LIN {X 0,Y 105.246,Z 1223.954,A -85,B 0,C 180,E1 5404.905,E2 5404.905} C_VEL
LIN {X 0,Y 105.222,Z 1230.827,A -85,B 0,C 180,E1 5396.186,E2 5396.186} C_VEL
LIN {X 0,Y 106.17,Z 1236.984,A -85,B 0,C 180,E1 5386.937,E2 5386.937} C_VEL
LIN {X 0,Y 110.756,Z 1244.43,A -85,B 0,C 180,E1 5373.745,E2 5373.745} C_VEL
LIN {X 0,Y 122.979,Z 1251.855,A -85,B 0,C 180,E1 5359.424,E2 5359.424} C_VEL
LIN {X 0,Y 127.608,Z 1253.595,A -85,B 0,C 180,E1 5355.812,E2 5355.812} C_VEL
LIN {X 0,Y 113.507,Z 1251.143,A -85,B 0,C 180,E1 5342.256,E2 5342.256} C_VEL
LIN {X 0,Y 107.747,Z 1247.277,A -85,B 0,C 180,E1 5327.84,E2 5327.84} C_VEL
LIN {X 0,Y 107.702,Z 1242.807,A -85,B 0,C 180,E1 5316.404,E2 5316.404} C_VEL
LIN {X 0,Y 108.21,Z 1239.966,A -85,B 0,C 180,E1 5311.066,E2 5311.066} C_VEL
LIN {X 0,Y 107.704,Z 1235.764,A -85,B 0,C 180,E1 5305.214,E2 5305.214} C_VEL
LIN {X 0,Y 106.691,Z 1233.424,A -85,B 0,C 180,E1 5296.458,E2 5296.458} C_VEL
LIN {X 0,Y 107.812,Z 1229.194,A -85,B 0,C 180,E1 5287.083,E2 5287.083} C_VEL
LIN {X 0,Y 111.454,Z 1223,A -85,B 0,C 180,E1 5278.05,E2 5278.05} C_VEL
LIN {X 0,Y 117.077,Z 1215.245,A -85,B 0,C 180,E1 5270.178,E2 5270.178} C_VEL
LIN {X 0,Y 124.096,Z 1206.072,A -85,B 0,C 180,E1 5263.528,E2 5263.528} C_VEL
LIN {X 0,Y 128.676,Z 1200.056,A -85,B 0,C 180,E1 5260.161,E2 5260.161} C_VEL
LIN {X 0,Y 131.324,Z 1195.46,A -85,B 0,C 180,E1 5257.692,E2 5257.692} C_VEL
LIN {X 0,Y 135.926,Z 1183.249,A -85,B 0,C 180,E1 5251.112,E2 5251.112} C_VEL
LIN {X 0,Y 138.939,Z 1177.877,A -85,B 0,C 180,E1 5249.119,E2 5249.119} C_VEL
LIN {X 0,Y 147.608,Z 1163.811,A -85,B 0,C 180,E1 5245.692,E2 5245.692} C_VEL
LIN {X 0,Y 155.785,Z 1148.222,A -85,B 0,C 180,E1 5242.936,E2 5242.936} C_VEL
LIN {X 0,Y 162.689,Z 1132.349,A -85,B 0,C 180,E1 5240.917,E2 5240.917} C_VEL
LIN {X 0,Y 168.161,Z 1116.222,A -85,B 0,C 180,E1 5239.397,E2 5239.397} C_VEL
LIN {X 0,Y 172.478,Z 1099.347,A -85,B 0,C 180,E1 5238.341,E2 5238.341} C_VEL
LIN {X 0,Y 175.176,Z 1083.244,A -85,B 0,C 180,E1 5237.612,E2 5237.612} C_VEL
LIN {X 0,Y 175.933,Z 1079.237,A -85,B 0,C 180,E1 5237.531,E2 5237.531} C_VEL
LIN {X 0,Y 193.961,Z 1045.169,A -85,B 0,C 180,E1 5234.022,E2 5234.022} C_VEL
LIN {X 0,Y 205.367,Z 1022.293,A -85,B 0,C 180,E1 5232.228,E2 5232.228} C_VEL
LIN {X 0,Y 209.325,Z 993.562,A -85,B 0,C 180,E1 5227.548,E2 5227.548} C_VEL
LIN {X 0,Y 214.843,Z 962.441,A -85,B 0,C 180,E1 5223.335,E2 5223.335} C_VEL
LIN {X 0,Y 220.959,Z 932.764,A -85,B 0,C 180,E1 5220.051,E2 5220.051} C_VEL
LIN {X 0,Y 225.837,Z 909.225,A -85,B 0,C 180,E1 5217.843,E2 5217.843} C_VEL
LIN {X 0,Y 221.843,Z 897.978,A -85,B 0,C 180,E1 5214.05,E2 5214.05} C_VEL
LIN {X 0,Y 217.917,Z 887.098,A -85,B 0,C 180,E1 5209.959,E2 5209.959} C_VEL
LIN {X 0,Y 214.165,Z 877.016,A -85,B 0,C 180,E1 5205.674,E2 5205.674} C_VEL
LIN {X 0,Y 210.547,Z 867.306,A -85,B 0,C 180,E1 5200.905,E2 5200.905} C_VEL
LIN {X 0,Y 208.954,Z 871.161,A -85,B 0,C 180,E1 5200.494,E2 5200.494} C_VEL
LIN {X 0,Y 201.666,Z 897.41,A -85,B 0,C 180,E1 5198.009,E2 5198.009} C_VEL
LIN {X 0,Y 201.281,Z 903.477,A -85,B 0,C 180,E1 5197.701,E2 5197.701} C_VEL
LIN {X 0,Y 187.356,Z 1041.59,A -85,B 0,C 180,E1 5194.545,E2 5194.545} C_VEL
LIN {X 0,Y 184.433,Z 1072.002,A -85,B 0,C 180,E1 5193.481,E2 5193.481} C_VEL
LIN {X 0,Y 181.214,Z 1089.478,A -85,B 0,C 180,E1 5192.503,E2 5192.503} C_VEL
LIN {X 0,Y 176.777,Z 1105.672,A -85,B 0,C 180,E1 5191.238,E2 5191.238} C_VEL
LIN {X 0,Y 171.003,Z 1121.455,A -85,B 0,C 180,E1 5189.584,E2 5189.584} C_VEL
LIN {X 0,Y 164.148,Z 1136.18,A -85,B 0,C 180,E1 5187.518,E2 5187.518} C_VEL
LIN {X 0,Y 155.96,Z 1150.576,A -85,B 0,C 180,E1 5184.818,E2 5184.818} C_VEL
LIN {X 0,Y 147,Z 1163.809,A -85,B 0,C 180,E1 5181.456,E2 5181.456} C_VEL
LIN {X 0,Y 138.159,Z 1174.954,A -85,B 0,C 180,E1 5177.569,E2 5177.569} C_VEL
LIN {X 0,Y 128.711,Z 1185.306,A -85,B 0,C 180,E1 5172.512,E2 5172.512} C_VEL
LIN {X 0,Y 119.744,Z 1194.066,A -85,B 0,C 180,E1 5166.352,E2 5166.352} C_VEL
LIN {X 0,Y 112.17,Z 1200.798,A -85,B 0,C 180,E1 5159.35,E2 5159.35} C_VEL
LIN {X 0,Y 105.944,Z 1205.962,A -85,B 0,C 180,E1 5151.009,E2 5151.009} C_VEL
LIN {X 0,Y 101.666,Z 1209.512,A -85,B 0,C 180,E1 5141.336,E2 5141.336} C_VEL
LIN {X 0,Y 99.952,Z 1211.169,A -85,B 0,C 180,E1 5131.712,E2 5131.712} C_VEL
LIN {X 0,Y 100.48,Z 1211.2,A -85,B 0,C 180,E1 5121.984,E2 5121.984} C_VEL
LIN {X 0,Y 103.519,Z 1209.445,A -85,B 0,C 180,E1 5111.988,E2 5111.988} C_VEL
LIN {X 0,Y 109.06,Z 1205.838,A -85,B 0,C 180,E1 5102.708,E2 5102.708} C_VEL
LIN {X 0,Y 116.376,Z 1200.564,A -85,B 0,C 180,E1 5094.847,E2 5094.847} C_VEL
LIN {X 0,Y 124.838,Z 1193.715,A -85,B 0,C 180,E1 5088.327,E2 5088.327} C_VEL
LIN {X 0,Y 127.493,Z 1191.387,A -85,B 0,C 180,E1 5086.539,E2 5086.539} C_VEL
LIN {X 0,Y 122.516,Z 1191.944,A -85,B 0,C 180,E1 5083.925,E2 5083.925} C_VEL
LIN {X 0,Y 116.388,Z 1192.651,A -85,B 0,C 180,E1 5080.115,E2 5080.115} C_VEL
LIN {X 0,Y 112.55,Z 1193.064,A -85,B 0,C 180,E1 5077.165,E2 5077.165} C_VEL
LIN {X 0,Y 107.91,Z 1193.718,A -85,B 0,C 180,E1 5073.141,E2 5073.141} C_VEL
LIN {X 0,Y 107.062,Z 1193.93,A -85,B 0,C 180,E1 5071.848,E2 5071.848} C_VEL
LIN {X 0,Y 100.882,Z 1207.438,A -85,B 0,C 180,E1 5060.905,E2 5060.905} C_VEL
LIN {X 0,Y 97.839,Z 1218.58,A -85,B 0,C 180,E1 5049.411,E2 5049.411} C_VEL
LIN {X 0,Y 97.295,Z 1226.633,A -85,B 0,C 180,E1 5039.411,E2 5039.411} C_VEL
LIN {X 0,Y 97.882,Z 1233.02,A -85,B 0,C 180,E1 5029.999,E2 5029.999} C_VEL
LIN {X 0,Y 100.999,Z 1240.281,A -85,B 0,C 180,E1 5017.288,E2 5017.288} C_VEL
LIN {X 0,Y 110.969,Z 1248.106,A -85,B 0,C 180,E1 5002.214,E2 5002.214} C_VEL
LIN {X 0,Y 118.291,Z 1251.374,A -85,B 0,C 180,E1 4995.809,E2 4995.809} C_VEL
LIN {X 0,Y 105.003,Z 1248.407,A -85,B 0,C 180,E1 4981.591,E2 4981.591} C_VEL
LIN {X 0,Y 99.966,Z 1243.981,A -85,B 0,C 180,E1 4966.215,E2 4966.215} C_VEL
LIN {X 0,Y 100.289,Z 1239.571,A -85,B 0,C 180,E1 4955.156,E2 4955.156} C_VEL
LIN {X 0,Y 100.561,Z 1237.068,A -85,B 0,C 180,E1 4950.577,E2 4950.577} C_VEL
LIN {X 0,Y 100.232,Z 1235.217,A -85,B 0,C 180,E1 4947.721,E2 4947.721} C_VEL
LIN {X 0,Y 98.773,Z 1233.364,A -85,B 0,C 180,E1 4938.327,E2 4938.327} C_VEL
LIN {X 0,Y 99.507,Z 1229.605,A -85,B 0,C 180,E1 4928.183,E2 4928.183} C_VEL
LIN {X 0,Y 102.95,Z 1223.987,A -85,B 0,C 180,E1 4918.377,E2 4918.377} C_VEL
LIN {X 0,Y 108.692,Z 1216.755,A -85,B 0,C 180,E1 4909.778,E2 4909.778} C_VEL
LIN {X 0,Y 116.303,Z 1207.694,A -85,B 0,C 180,E1 4902.333,E2 4902.333} C_VEL
LIN {X 0,Y 125.095,Z 1196.89,A -85,B 0,C 180,E1 4896.179,E2 4896.179} C_VEL
LIN {X 0,Y 133.685,Z 1185.442,A -85,B 0,C 180,E1 4891.511,E2 4891.511} C_VEL
LIN {X 0,Y 138.939,Z 1177.877,A -85,B 0,C 180,E1 4889.119,E2 4889.119} C_VEL
LIN {X 0,Y 142.011,Z 1172.369,A -85,B 0,C 180,E1 4887.266,E2 4887.266} C_VEL
LIN {X 0,Y 147.233,Z 1158.819,A -85,B 0,C 180,E1 4882.408,E2 4882.408} C_VEL
LIN {X 0,Y 149.975,Z 1152.651,A -85,B 0,C 180,E1 4880.934,E2 4880.934} C_VEL
LIN {X 0,Y 150.44,Z 1151.73,A -85,B 0,C 180,E1 4880.778,E2 4880.778} C_VEL
LIN {X 0,Y 157.803,Z 1136.272,A -85,B 0,C 180,E1 4878.705,E2 4878.705} C_VEL
LIN {X 0,Y 163.802,Z 1120.734,A -85,B 0,C 180,E1 4877.212,E2 4877.212} C_VEL
LIN {X 0,Y 168.776,Z 1103.64,A -85,B 0,C 180,E1 4875.989,E2 4875.989} C_VEL
LIN {X 0,Y 172.33,Z 1086.034,A -85,B 0,C 180,E1 4875.19,E2 4875.19} C_VEL
LIN {X 0,Y 174.295,Z 1070.714,A -85,B 0,C 180,E1 4874.86,E2 4874.86} C_VEL
LIN {X 0,Y 192.293,Z 1037.002,A -85,B 0,C 180,E1 4871.7,E2 4871.7} C_VEL
LIN {X 0,Y 199.398,Z 1022.993,A -85,B 0,C 180,E1 4870.652,E2 4870.652} C_VEL
LIN {X 0,Y 203.623,Z 995.232,A -85,B 0,C 180,E1 4866.06,E2 4866.06} C_VEL
LIN {X 0,Y 209.363,Z 965.34,A -85,B 0,C 180,E1 4861.916,E2 4861.916} C_VEL
LIN {X 0,Y 215.887,Z 935.47,A -85,B 0,C 180,E1 4858.54,E2 4858.54} C_VEL
LIN {X 0,Y 220.861,Z 913.307,A -85,B 0,C 180,E1 4856.431,E2 4856.431} C_VEL
LIN {X 0,Y 216.303,Z 899.981,A -85,B 0,C 180,E1 4851.761,E2 4851.761} C_VEL
LIN {X 0,Y 211.472,Z 886.05,A -85,B 0,C 180,E1 4846.046,E2 4846.046} C_VEL
LIN {X 0,Y 208.474,Z 877.998,A -85,B 0,C 180,E1 4842.171,E2 4842.171} C_VEL
LIN {X 0,Y 199.404,Z 895.735,A -85,B 0,C 180,E1 4840.369,E2 4840.369} C_VEL
LIN {X 0,Y 198.806,Z 899.822,A -85,B 0,C 180,E1 4840.046,E2 4840.046} C_VEL
LIN {X 0,Y 198.303,Z 905.835,A -85,B 0,C 180,E1 4839.811,E2 4839.811} C_VEL
LIN {X 0,Y 184.18,Z 1042.051,A -85,B 0,C 180,E1 4836.805,E2 4836.805} C_VEL
LIN {X 0,Y 181.08,Z 1072.972,A -85,B 0,C 180,E1 4835.741,E2 4835.741} C_VEL
LIN {X 0,Y 177.72,Z 1090.534,A -85,B 0,C 180,E1 4834.779,E2 4834.779} C_VEL
LIN {X 0,Y 173.102,Z 1106.793,A -85,B 0,C 180,E1 4833.539,E2 4833.539} C_VEL
LIN {X 0,Y 167.128,Z 1122.537,A -85,B 0,C 180,E1 4831.929,E2 4831.929} C_VEL
LIN {X 0,Y 160.029,Z 1137.233,A -85,B 0,C 180,E1 4829.914,E2 4829.914} C_VEL
LIN {X 0,Y 151.528,Z 1151.613,A -85,B 0,C 180,E1 4827.27,E2 4827.27} C_VEL
LIN {X 0,Y 142.191,Z 1164.833,A -85,B 0,C 180,E1 4823.957,E2 4823.957} C_VEL
LIN {X 0,Y 132.932,Z 1175.961,A -85,B 0,C 180,E1 4820.095,E2 4820.095} C_VEL
LIN {X 0,Y 122.976,Z 1186.305,A -85,B 0,C 180,E1 4815.012,E2 4815.012} C_VEL
LIN {X 0,Y 113.446,Z 1195.056,A -85,B 0,C 180,E1 4808.73,E2 4808.73} C_VEL
LIN {X 0,Y 105.318,Z 1201.777,A -85,B 0,C 180,E1 4801.469,E2 4801.469} C_VEL
LIN {X 0,Y 98.571,Z 1206.934,A -85,B 0,C 180,E1 4792.664,E2 4792.664} C_VEL
LIN {X 0,Y 93.892,Z 1210.477,A -85,B 0,C 180,E1 4782.289,E2 4782.289} C_VEL
LIN {X 0,Y 92.013,Z 1212.127,A -85,B 0,C 180,E1 4771.86,E2 4771.86} C_VEL
LIN {X 0,Y 92.615,Z 1212.148,A -85,B 0,C 180,E1 4761.298,E2 4761.298} C_VEL
LIN {X 0,Y 95.985,Z 1210.386,A -85,B 0,C 180,E1 4750.52,E2 4750.52} C_VEL
LIN {X 0,Y 102.051,Z 1206.773,A -85,B 0,C 180,E1 4740.658,E2 4740.658} C_VEL
LIN {X 0,Y 109.961,Z 1201.487,A -85,B 0,C 180,E1 4732.457,E2 4732.457} C_VEL
LIN {X 0,Y 117.792,Z 1195.575,A -85,B 0,C 180,E1 4726.471,E2 4726.471} C_VEL
LIN {X 0,Y 106.932,Z 1196.858,A -85,B 0,C 180,E1 4719.483,E2 4719.483} C_VEL
LIN {X 0,Y 101.589,Z 1197.56,A -85,B 0,C 180,E1 4714.811,E2 4714.811} C_VEL
LIN {X 0,Y 99.608,Z 1197.869,A -85,B 0,C 180,E1 4712.824,E2 4712.824} C_VEL
LIN {X 0,Y 96.735,Z 1198.241,A -85,B 0,C 180,E1 4709.066,E2 4709.066} C_VEL
LIN {X 0,Y 96.47,Z 1198.357,A -85,B 0,C 180,E1 4708.476,E2 4708.476} C_VEL
LIN {X 0,Y 91.408,Z 1210.905,A -85,B 0,C 180,E1 4696.524,E2 4696.524} C_VEL
LIN {X 0,Y 89.577,Z 1220.487,A -85,B 0,C 180,E1 4685.123,E2 4685.123} C_VEL
LIN {X 0,Y 89.671,Z 1227.741,A -85,B 0,C 180,E1 4674.882,E2 4674.882} C_VEL
LIN {X 0,Y 91.049,Z 1234.203,A -85,B 0,C 180,E1 4664.065,E2 4664.065} C_VEL
LIN {X 0,Y 97.502,Z 1242.365,A -85,B 0,C 180,E1 4648.353,E2 4648.353} C_VEL
LIN {X 0,Y 108.975,Z 1248.805,A -85,B 0,C 180,E1 4635.709,E2 4635.709} C_VEL
LIN {X 0,Y 96.178,Z 1245.153,A -85,B 0,C 180,E1 4619.944,E2 4619.944} C_VEL
LIN {X 0,Y 92.311,Z 1240.244,A -85,B 0,C 180,E1 4603.795,E2 4603.795} C_VEL
LIN {X 0,Y 92.93,Z 1236.108,A -85,B 0,C 180,E1 4593.71,E2 4593.71} C_VEL
LIN {X 0,Y 92.901,Z 1234.458,A -85,B 0,C 180,E1 4590.625,E2 4590.625} C_VEL
LIN {X 0,Y 91.048,Z 1233.235,A -85,B 0,C 180,E1 4581.165,E2 4581.165} C_VEL
LIN {X 0,Y 91.136,Z 1230.116,A -85,B 0,C 180,E1 4570.126,E2 4570.126} C_VEL
LIN {X 0,Y 94.245,Z 1225.111,A -85,B 0,C 180,E1 4559.246,E2 4559.246} C_VEL
LIN {X 0,Y 99.706,Z 1218.754,A -85,B 0,C 180,E1 4550.084,E2 4550.084} C_VEL
LIN {X 0,Y 107.448,Z 1210.335,A -85,B 0,C 180,E1 4541.899,E2 4541.899} C_VEL
LIN {X 0,Y 116.421,Z 1200.433,A -85,B 0,C 180,E1 4535.335,E2 4535.335} C_VEL
LIN {X 0,Y 126.065,Z 1188.866,A -85,B 0,C 180,E1 4529.98,E2 4529.98} C_VEL
LIN {X 0,Y 135.538,Z 1176.14,A -85,B 0,C 180,E1 4525.854,E2 4525.854} C_VEL
LIN {X 0,Y 144.574,Z 1162.104,A -85,B 0,C 180,E1 4522.603,E2 4522.603} C_VEL
LIN {X 0,Y 150.44,Z 1151.73,A -85,B 0,C 180,E1 4520.778,E2 4520.778} C_VEL
LIN {X 0,Y 153.253,Z 1145.34,A -85,B 0,C 180,E1 4519.468,E2 4519.468} C_VEL
LIN {X 0,Y 158.065,Z 1130.034,A -85,B 0,C 180,E1 4515.698,E2 4515.698} C_VEL
LIN {X 0,Y 160.316,Z 1123.16,A -85,B 0,C 180,E1 4514.714,E2 4514.714} C_VEL
LIN {X 0,Y 160.679,Z 1122.139,A -85,B 0,C 180,E1 4514.635,E2 4514.635} C_VEL
LIN {X 0,Y 165.933,Z 1105.428,A -85,B 0,C 180,E1 4513.463,E2 4513.463} C_VEL
LIN {X 0,Y 169.833,Z 1087.915,A -85,B 0,C 180,E1 4512.69,E2 4512.69} C_VEL
LIN {X 0,Y 172.131,Z 1071.306,A -85,B 0,C 180,E1 4512.294,E2 4512.294} C_VEL
LIN {X 0,Y 173.184,Z 1061.961,A -85,B 0,C 180,E1 4512.119,E2 4512.119} C_VEL
LIN {X 0,Y 193.352,Z 1023.934,A -85,B 0,C 180,E1 4509.017,E2 4509.017} C_VEL
LIN {X 0,Y 198.599,Z 993.903,A -85,B 0,C 180,E1 4504.042,E2 4504.042} C_VEL
LIN {X 0,Y 205.211,Z 962.503,A -85,B 0,C 180,E1 4499.721,E2 4499.721} C_VEL
LIN {X 0,Y 212.392,Z 931.815,A -85,B 0,C 180,E1 4496.344,E2 4496.344} C_VEL
LIN {X 0,Y 215.793,Z 917.203,A -85,B 0,C 180,E1 4494.949,E2 4494.949} C_VEL
LIN {X 0,Y 211.105,Z 902.797,A -85,B 0,C 180,E1 4489.631,E2 4489.631} C_VEL
LIN {X 0,Y 206.97,Z 890.424,A -85,B 0,C 180,E1 4484.303,E2 4484.303} C_VEL
LIN {X 0,Y 206.369,Z 888.736,A -85,B 0,C 180,E1 4483.467,E2 4483.467} C_VEL
LIN {X 0,Y 200.384,Z 899.887,A -85,B 0,C 180,E1 4482.361,E2 4482.361} C_VEL
LIN {X 0,Y 195.246,Z 911.483,A -85,B 0,C 180,E1 4481.919,E2 4481.919} C_VEL
LIN {X 0,Y 181.301,Z 1042.512,A -85,B 0,C 180,E1 4479.141,E2 4479.141} C_VEL
LIN {X 0,Y 178.044,Z 1073.784,A -85,B 0,C 180,E1 4478.09,E2 4478.09} C_VEL
LIN {X 0,Y 174.591,Z 1091.291,A -85,B 0,C 180,E1 4477.161,E2 4477.161} C_VEL
LIN {X 0,Y 169.717,Z 1107.91,A -85,B 0,C 180,E1 4475.936,E2 4475.936} C_VEL
LIN {X 0,Y 163.546,Z 1123.615,A -85,B 0,C 180,E1 4474.381,E2 4474.381} C_VEL
LIN {X 0,Y 155.798,Z 1138.998,A -85,B 0,C 180,E1 4472.321,E2 4472.321} C_VEL
LIN {X 0,Y 146.996,Z 1153.238,A -85,B 0,C 180,E1 4469.743,E2 4469.743} C_VEL
LIN {X 0,Y 137.672,Z 1165.856,A -85,B 0,C 180,E1 4466.628,E2 4466.628} C_VEL
LIN {X 0,Y 127.986,Z 1176.968,A -85,B 0,C 180,E1 4462.822,E2 4462.822} C_VEL
LIN {X 0,Y 117.547,Z 1187.258,A -85,B 0,C 180,E1 4457.778,E2 4457.778} C_VEL
LIN {X 0,Y 107.367,Z 1196.047,A -85,B 0,C 180,E1 4451.382,E2 4451.382} C_VEL
LIN {X 0,Y 98.631,Z 1202.756,A -85,B 0,C 180,E1 4443.878,E2 4443.878} C_VEL
LIN {X 0,Y 91.292,Z 1207.906,A -85,B 0,C 180,E1 4434.585,E2 4434.585} C_VEL
LIN {X 0,Y 86.148,Z 1211.442,A -85,B 0,C 180,E1 4423.413,E2 4423.413} C_VEL
LIN {X 0,Y 84.075,Z 1213.085,A -85,B 0,C 180,E1 4412.035,E2 4412.035} C_VEL
LIN {X 0,Y 84.766,Z 1213.096,A -85,B 0,C 180,E1 4400.485,E2 4400.485} C_VEL
LIN {X 0,Y 88.524,Z 1211.328,A -85,B 0,C 180,E1 4388.802,E2 4388.802} C_VEL
LIN {X 0,Y 95.221,Z 1207.691,A -85,B 0,C 180,E1 4378.273,E2 4378.273} C_VEL
LIN {X 0,Y 103.761,Z 1202.41,A -85,B 0,C 180,E1 4369.777,E2 4369.777} C_VEL
LIN {X 0,Y 107.976,Z 1199.5,A -85,B 0,C 180,E1 4366.457,E2 4366.457} C_VEL
LIN {X 0,Y 95.233,Z 1201.084,A -85,B 0,C 180,E1 4356.761,E2 4356.761} C_VEL
LIN {X 0,Y 90.408,Z 1201.81,A -85,B 0,C 180,E1 4351.32,E2 4351.32} C_VEL
LIN {X 0,Y 86.45,Z 1202.554,A -85,B 0,C 180,E1 4345.337,E2 4345.337} C_VEL
LIN {X 0,Y 86.004,Z 1202.856,A -85,B 0,C 180,E1 4344.011,E2 4344.011} C_VEL
LIN {X 0,Y 82.397,Z 1214.068,A -85,B 0,C 180,E1 4331.196,E2 4331.196} C_VEL
LIN {X 0,Y 81.703,Z 1222.661,A -85,B 0,C 180,E1 4319.299,E2 4319.299} C_VEL
LIN {X 0,Y 82.475,Z 1229.04,A -85,B 0,C 180,E1 4308.815,E2 4308.815} C_VEL
LIN {X 0,Y 86.1,Z 1236.489,A -85,B 0,C 180,E1 4294.552,E2 4294.552} C_VEL
LIN {X 0,Y 97.252,Z 1244.659,A -85,B 0,C 180,E1 4278.064,E2 4278.064} C_VEL
LIN {X 0,Y 99.764,Z 1245.912,A -85,B 0,C 180,E1 4275.58,E2 4275.58} C_VEL
LIN {X 0,Y 87.88,Z 1241.76,A -85,B 0,C 180,E1 4258.825,E2 4258.825} C_VEL
LIN {X 0,Y 84.851,Z 1236.588,A -85,B 0,C 180,E1 4242.018,E2 4242.018} C_VEL
LIN {X 0,Y 85.367,Z 1233.541,A -85,B 0,C 180,E1 4234.039,E2 4234.039} C_VEL
LIN {X 0,Y 84.538,Z 1233.408,A -85,B 0,C 180,E1 4229.332,E2 4229.332} C_VEL
LIN {X 0,Y 82.822,Z 1231.821,A -85,B 0,C 180,E1 4218.166,E2 4218.166} C_VEL
LIN {X 0,Y 83.84,Z 1228.399,A -85,B 0,C 180,E1 4206.089,E2 4206.089} C_VEL
LIN {X 0,Y 88.134,Z 1223.096,A -85,B 0,C 180,E1 4194.659,E2 4194.659} C_VEL
LIN {X 0,Y 95.374,Z 1215.821,A -85,B 0,C 180,E1 4184.622,E2 4184.622} C_VEL
LIN {X 0,Y 104.526,Z 1206.871,A -85,B 0,C 180,E1 4176.544,E2 4176.544} C_VEL
LIN {X 0,Y 114.094,Z 1196.956,A -85,B 0,C 180,E1 4170.551,E2 4170.551} C_VEL
LIN {X 0,Y 124.259,Z 1185.23,A -85,B 0,C 180,E1 4165.694,E2 4165.694} C_VEL
LIN {X 0,Y 134.578,Z 1171.658,A -85,B 0,C 180,E1 4161.781,E2 4161.781} C_VEL
LIN {X 0,Y 143.739,Z 1157.63,A -85,B 0,C 180,E1 4158.924,E2 4158.924} C_VEL
LIN {X 0,Y 151.886,Z 1142.615,A -85,B 0,C 180,E1 4156.715,E2 4156.715} C_VEL
LIN {X 0,Y 158.881,Z 1126.721,A -85,B 0,C 180,E1 4155,E2 4155} C_VEL
LIN {X 0,Y 160.679,Z 1122.139,A -85,B 0,C 180,E1 4154.635,E2 4154.635} C_VEL
LIN {X 0,Y 162.91,Z 1115.059,A -85,B 0,C 180,E1 4153.844,E2 4153.844} C_VEL
LIN {X 0,Y 166.41,Z 1097.259,A -85,B 0,C 180,E1 4150.852,E2 4150.852} C_VEL
LIN {X 0,Y 167.652,Z 1089.886,A -85,B 0,C 180,E1 4150.133,E2 4150.133} C_VEL
LIN {X 0,Y 170.211,Z 1072.999,A -85,B 0,C 180,E1 4149.669,E2 4149.669} C_VEL
LIN {X 0,Y 172.581,Z 1052.632,A -85,B 0,C 180,E1 4149.363,E2 4149.363} C_VEL
LIN {X 0,Y 187.818,Z 1023.896,A -85,B 0,C 180,E1 4147.202,E2 4147.202} C_VEL
LIN {X 0,Y 193.583,Z 993.414,A -85,B 0,C 180,E1 4142.072,E2 4142.072} C_VEL
LIN {X 0,Y 200.964,Z 960.888,A -85,B 0,C 180,E1 4137.623,E2 4137.623} C_VEL
LIN {X 0,Y 208.275,Z 931.485,A -85,B 0,C 180,E1 4134.421,E2 4134.421} C_VEL
LIN {X 0,Y 210.778,Z 921.02,A -85,B 0,C 180,E1 4133.394,E2 4133.394} C_VEL
LIN {X 0,Y 206.432,Z 907.03,A -85,B 0,C 180,E1 4127.978,E2 4127.978} C_VEL
LIN {X 0,Y 204.057,Z 899.506,A -85,B 0,C 180,E1 4124.713,E2 4124.713} C_VEL
LIN {X 0,Y 201.441,Z 904.601,A -85,B 0,C 180,E1 4124.338,E2 4124.338} C_VEL
LIN {X 0,Y 197.022,Z 914.385,A -85,B 0,C 180,E1 4124.13,E2 4124.13} C_VEL
LIN {X 0,Y 192.414,Z 924.63,A -85,B 0,C 180,E1 4124.003,E2 4124.003} C_VEL
LIN {X 0,Y 191.311,Z 927.505,A -85,B 0,C 180,E1 4123.9,E2 4123.9} C_VEL
LIN {X 0,Y 178.706,Z 1043.23,A -85,B 0,C 180,E1 4121.541,E2 4121.541} C_VEL
LIN {X 0,Y 175.292,Z 1074.749,A -85,B 0,C 180,E1 4120.509,E2 4120.509} C_VEL
LIN {X 0,Y 171.722,Z 1092.254,A -85,B 0,C 180,E1 4119.614,E2 4119.614} C_VEL
LIN {X 0,Y 166.641,Z 1109.029,A -85,B 0,C 180,E1 4118.426,E2 4118.426} C_VEL
LIN {X 0,Y 160.277,Z 1124.691,A -85,B 0,C 180,E1 4116.938,E2 4116.938} C_VEL
LIN {X 0,Y 152.276,Z 1140.048,A -85,B 0,C 180,E1 4114.965,E2 4114.965} C_VEL
LIN {X 0,Y 143.163,Z 1154.273,A -85,B 0,C 180,E1 4112.486,E2 4112.486} C_VEL
LIN {X 0,Y 133.472,Z 1166.878,A -85,B 0,C 180,E1 4109.474,E2 4109.474} C_VEL
LIN {X 0,Y 123.351,Z 1177.974,A -85,B 0,C 180,E1 4105.761,E2 4105.761} C_VEL
LIN {X 0,Y 112.313,Z 1188.3,A -85,B 0,C 180,E1 4100.751,E2 4100.751} C_VEL
LIN {X 0,Y 101.544,Z 1197.036,A -85,B 0,C 180,E1 4094.346,E2 4094.346} C_VEL
LIN {X 0,Y 92.143,Z 1203.735,A -85,B 0,C 180,E1 4086.632,E2 4086.632} C_VEL
LIN {X 0,Y 84.133,Z 1208.878,A -85,B 0,C 180,E1 4076.836,E2 4076.836} C_VEL
LIN {X 0,Y 78.444,Z 1212.406,A -85,B 0,C 180,E1 4064.759,E2 4064.759} C_VEL
LIN {X 0,Y 76.138,Z 1214.043,A -85,B 0,C 180,E1 4052.248,E2 4052.248} C_VEL
LIN {X 0,Y 76.937,Z 1214.045,A -85,B 0,C 180,E1 4039.507,E2 4039.507} C_VEL
LIN {X 0,Y 81.157,Z 1212.271,A -85,B 0,C 180,E1 4026.77,E2 4026.77} C_VEL
LIN {X 0,Y 88.517,Z 1208.643,A -85,B 0,C 180,E1 4015.601,E2 4015.601} C_VEL
LIN {X 0,Y 97.816,Z 1203.333,A -85,B 0,C 180,E1 4006.764,E2 4006.764} C_VEL
LIN {X 0,Y 97.944,Z 1203.175,A -85,B 0,C 180,E1 4006.455,E2 4006.455} C_VEL
LIN {X 0,Y 83.56,Z 1205.08,A -85,B 0,C 180,E1 3992.988,E2 3992.988} C_VEL
LIN {X 0,Y 79.814,Z 1205.81,A -85,B 0,C 180,E1 3987.615,E2 3987.615} C_VEL
LIN {X 0,Y 78.383,Z 1206.122,A -85,B 0,C 180,E1 3984.896,E2 3984.896} C_VEL
LIN {X 0,Y 76.113,Z 1206.716,A -85,B 0,C 180,E1 3978.676,E2 3978.676} C_VEL
LIN {X 0,Y 74.015,Z 1216.443,A -85,B 0,C 180,E1 3965.426,E2 3965.426} C_VEL
LIN {X 0,Y 74.252,Z 1223.648,A -85,B 0,C 180,E1 3953.816,E2 3953.816} C_VEL
LIN {X 0,Y 76.009,Z 1230.082,A -85,B 0,C 180,E1 3941.596,E2 3941.596} C_VEL
LIN {X 0,Y 83.953,Z 1238.752,A -85,B 0,C 180,E1 3923.451,E2 3923.451} C_VEL
LIN {X 0,Y 90.647,Z 1242.703,A -85,B 0,C 180,E1 3915.386,E2 3915.386} C_VEL
LIN {X 0,Y 79.463,Z 1237.897,A -85,B 0,C 180,E1 3896.696,E2 3896.696} C_VEL
LIN {X 0,Y 77.565,Z 1232.484,A -85,B 0,C 180,E1 3879.283,E2 3879.283} C_VEL
LIN {X 0,Y 77.299,Z 1232.622,A -85,B 0,C 180,E1 3872.976,E2 3872.976} C_VEL
LIN {X 0,Y 75.319,Z 1231.835,A -85,B 0,C 180,E1 3863.149,E2 3863.149} C_VEL
LIN {X 0,Y 75.156,Z 1229.235,A -85,B 0,C 180,E1 3849.774,E2 3849.774} C_VEL
LIN {X 0,Y 78.636,Z 1224.817,A -85,B 0,C 180,E1 3836.867,E2 3836.867} C_VEL
LIN {X 0,Y 85.529,Z 1218.446,A -85,B 0,C 180,E1 3825.471,E2 3825.471} C_VEL
LIN {X 0,Y 94.54,Z 1210.544,A -85,B 0,C 180,E1 3816.52,E2 3816.52} C_VEL
LIN {X 0,Y 104.719,Z 1201.225,A -85,B 0,C 180,E1 3809.686,E2 3809.686} C_VEL
LIN {X 0,Y 115.272,Z 1190.448,A -85,B 0,C 180,E1 3804.404,E2 3804.404} C_VEL
LIN {X 0,Y 126.23,Z 1177.713,A -85,B 0,C 180,E1 3800.193,E2 3800.193} C_VEL
LIN {X 0,Y 136.317,Z 1164.093,A -85,B 0,C 180,E1 3797.062,E2 3797.062} C_VEL
LIN {X 0,Y 145.077,Z 1150.128,A -85,B 0,C 180,E1 3794.774,E2 3794.774} C_VEL
LIN {X 0,Y 152.889,Z 1135.048,A -85,B 0,C 180,E1 3793.005,E2 3793.005} C_VEL
LIN {X 0,Y 159.263,Z 1119.705,A -85,B 0,C 180,E1 3791.677,E2 3791.677} C_VEL
LIN {X 0,Y 164.718,Z 1102.479,A -85,B 0,C 180,E1 3790.638,E2 3790.638} C_VEL
LIN {X 0,Y 167.652,Z 1089.886,A -85,B 0,C 180,E1 3790.133,E2 3790.133} C_VEL
LIN {X 0,Y 168.717,Z 1082.401,A -85,B 0,C 180,E1 3789.47,E2 3789.47} C_VEL
LIN {X 0,Y 170.002,Z 1064.702,A -85,B 0,C 180,E1 3787.18,E2 3787.18} C_VEL
LIN {X 0,Y 170.716,Z 1057.143,A -85,B 0,C 180,E1 3786.714,E2 3786.714} C_VEL
LIN {X 0,Y 170.845,Z 1056.048,A -85,B 0,C 180,E1 3786.701,E2 3786.701} C_VEL
LIN {X 0,Y 172.607,Z 1042.08,A -85,B 0,C 180,E1 3786.595,E2 3786.595} C_VEL
LIN {X 0,Y 182.185,Z 1024.297,A -85,B 0,C 180,E1 3785.354,E2 3785.354} C_VEL
LIN {X 0,Y 188.523,Z 993.699,A -85,B 0,C 180,E1 3780.152,E2 3780.152} C_VEL
LIN {X 0,Y 195.992,Z 962.973,A -85,B 0,C 180,E1 3775.904,E2 3775.904} C_VEL
LIN {X 0,Y 204.212,Z 931.471,A -85,B 0,C 180,E1 3772.474,E2 3772.474} C_VEL
LIN {X 0,Y 205.871,Z 925.076,A -85,B 0,C 180,E1 3771.833,E2 3771.833} C_VEL
LIN {X 0,Y 202.135,Z 912.54,A -85,B 0,C 180,E1 3766.847,E2 3766.847} C_VEL
LIN {X 0,Y 201.695,Z 911.437,A -85,B 0,C 180,E1 3766.307,E2 3766.307} C_VEL
LIN {X 0,Y 195.11,Z 926.263,A -85,B 0,C 180,E1 3766.181,E2 3766.181} C_VEL
LIN {X 0,Y 188.524,Z 940.406,A -85,B 0,C 180,E1 3766.05,E2 3766.05} C_VEL
LIN {X 0,Y 187.7,Z 942.755,A -85,B 0,C 180,E1 3765.976,E2 3765.976} C_VEL
LIN {X 0,Y 176.405,Z 1044.225,A -85,B 0,C 180,E1 3764,E2 3764} C_VEL
LIN {X 0,Y 172.862,Z 1075.714,A -85,B 0,C 180,E1 3763.001,E2 3763.001} C_VEL
LIN {X 0,Y 169.162,Z 1093.276,A -85,B 0,C 180,E1 3762.141,E2 3762.141} C_VEL
LIN {X 0,Y 163.892,Z 1110.149,A -85,B 0,C 180,E1 3761.005,E2 3761.005} C_VEL
LIN {X 0,Y 157.34,Z 1125.766,A -85,B 0,C 180,E1 3759.596,E2 3759.596} C_VEL
LIN {X 0,Y 149.093,Z 1141.099,A -85,B 0,C 180,E1 3757.728,E2 3757.728} C_VEL
LIN {X 0,Y 139.675,Z 1155.308,A -85,B 0,C 180,E1 3755.373,E2 3755.373} C_VEL
LIN {X 0,Y 129.622,Z 1167.899,A -85,B 0,C 180,E1 3752.496,E2 3752.496} C_VEL
LIN {X 0,Y 119.067,Z 1178.98,A -85,B 0,C 180,E1 3748.919,E2 3748.919} C_VEL
LIN {X 0,Y 107.466,Z 1189.298,A -85,B 0,C 180,E1 3744.031,E2 3744.031} C_VEL
LIN {X 0,Y 96.025,Z 1198.026,A -85,B 0,C 180,E1 3737.66,E2 3737.66} C_VEL
LIN {X 0,Y 85.899,Z 1204.713,A -85,B 0,C 180,E1 3729.795,E2 3729.795} C_VEL
LIN {X 0,Y 77.129,Z 1209.849,A -85,B 0,C 180,E1 3719.501,E2 3719.501} C_VEL
LIN {X 0,Y 70.793,Z 1213.371,A -85,B 0,C 180,E1 3706.397,E2 3706.397} C_VEL
LIN {X 0,Y 68.202,Z 1215.001,A -85,B 0,C 180,E1 3692.509,E2 3692.509} C_VEL
LIN {X 0,Y 69.136,Z 1214.993,A -85,B 0,C 180,E1 3678.307,E2 3678.307} C_VEL
LIN {X 0,Y 73.912,Z 1213.213,A -85,B 0,C 180,E1 3664.337,E2 3664.337} C_VEL
LIN {X 0,Y 82.071,Z 1209.578,A -85,B 0,C 180,E1 3652.46,E2 3652.46} C_VEL
LIN {X 0,Y 88.164,Z 1206.46,A -85,B 0,C 180,E1 3646.539,E2 3646.539} C_VEL
LIN {X 0,Y 71.257,Z 1209.123,A -85,B 0,C 180,E1 3626.682,E2 3626.682} C_VEL
LIN {X 0,Y 68.247,Z 1209.959,A -85,B 0,C 180,E1 3618.804,E2 3618.804} C_VEL
LIN {X 0,Y 66.713,Z 1210.924,A -85,B 0,C 180,E1 3610.798,E2 3610.798} C_VEL
LIN {X 0,Y 66.352,Z 1219.543,A -85,B 0,C 180,E1 3596.544,E2 3596.544} C_VEL
LIN {X 0,Y 67.671,Z 1225.652,A -85,B 0,C 180,E1 3584.576,E2 3584.576} C_VEL
LIN {X 0,Y 73.429,Z 1233.657,A -85,B 0,C 180,E1 3566.997,E2 3566.997} C_VEL
LIN {X 0,Y 81.735,Z 1239.176,A -85,B 0,C 180,E1 3555.21,E2 3555.21} C_VEL
LIN {X 0,Y 71.328,Z 1233.792,A -85,B 0,C 180,E1 3534.33,E2 3534.33} C_VEL
LIN {X 0,Y 70.037,Z 1230.991,A -85,B 0,C 180,E1 3523.877,E2 3523.877} C_VEL
LIN {X 0,Y 69.462,Z 1231.654,A -85,B 0,C 180,E1 3514.139,E2 3514.139} C_VEL
LIN {X 0,Y 67.317,Z 1230.944,A -85,B 0,C 180,E1 3503.187,E2 3503.187} C_VEL
LIN {X 0,Y 67.331,Z 1228.422,A -85,B 0,C 180,E1 3488.22,E2 3488.22} C_VEL
LIN {X 0,Y 71.455,Z 1224.12,A -85,B 0,C 180,E1 3474.019,E2 3474.019} C_VEL
LIN {X 0,Y 79.248,Z 1217.854,A -85,B 0,C 180,E1 3461.907,E2 3461.907} C_VEL
LIN {X 0,Y 89.832,Z 1209.506,A -85,B 0,C 180,E1 3452.245,E2 3452.245} C_VEL
LIN {X 0,Y 100.853,Z 1200.179,A -85,B 0,C 180,E1 3445.57,E2 3445.57} C_VEL
LIN {X 0,Y 112.092,Z 1189.389,A -85,B 0,C 180,E1 3440.529,E2 3440.529} C_VEL
LIN {X 0,Y 123.494,Z 1176.784,A -85,B 0,C 180,E1 3436.615,E2 3436.615} C_VEL
LIN {X 0,Y 134.264,Z 1162.828,A -85,B 0,C 180,E1 3433.653,E2 3433.653} C_VEL
LIN {X 0,Y 143.377,Z 1148.747,A -85,B 0,C 180,E1 3431.56,E2 3431.56} C_VEL
LIN {X 0,Y 151.551,Z 1133.29,A -85,B 0,C 180,E1 3429.922,E2 3429.922} C_VEL
LIN {X 0,Y 158.278,Z 1117.271,A -85,B 0,C 180,E1 3428.677,E2 3428.677} C_VEL
LIN {X 0,Y 163.439,Z 1101.235,A -85,B 0,C 180,E1 3427.861,E2 3427.861} C_VEL
LIN {X 0,Y 167.383,Z 1083.445,A -85,B 0,C 180,E1 3427.212,E2 3427.212} C_VEL
LIN {X 0,Y 170.845,Z 1056.048,A -85,B 0,C 180,E1 3426.701,E2 3426.701} C_VEL
LIN {X 0,Y 171.266,Z 1051.648,A -85,B 0,C 180,E1 3426.397,E2 3426.397} C_VEL
LIN {X 0,Y 172.134,Z 1038.106,A -85,B 0,C 180,E1 3424.045,E2 3424.045} C_VEL
LIN {X 0,Y 172.613,Z 1033.721,A -85,B 0,C 180,E1 3423.823,E2 3423.823} C_VEL
LIN {X 0,Y 173.078,Z 1031.394,A -85,B 0,C 180,E1 3423.848,E2 3423.848} C_VEL
LIN {X 0,Y 176.738,Z 1024.395,A -85,B 0,C 180,E1 3423.358,E2 3423.358} C_VEL
LIN {X 0,Y 183.652,Z 993.856,A -85,B 0,C 180,E1 3418.128,E2 3418.128} C_VEL
LIN {X 0,Y 191.988,Z 961.834,A -85,B 0,C 180,E1 3413.721,E2 3413.721} C_VEL
LIN {X 0,Y 200.89,Z 929.063,A -85,B 0,C 180,E1 3410.206,E2 3410.206} C_VEL
LIN {X 0,Y 199.57,Z 924.644,A -85,B 0,C 180,E1 3408.356,E2 3408.356} C_VEL
LIN {X 0,Y 196.034,Z 932.174,A -85,B 0,C 180,E1 3408.301,E2 3408.301} C_VEL
LIN {X 0,Y 190.979,Z 942.836,A -85,B 0,C 180,E1 3408.229,E2 3408.229} C_VEL
LIN {X 0,Y 185.862,Z 953.476,A -85,B 0,C 180,E1 3408.244,E2 3408.244} C_VEL
LIN {X 0,Y 184.503,Z 956.643,A -85,B 0,C 180,E1 3408.153,E2 3408.153} C_VEL
LIN {X 0,Y 174.428,Z 1045.299,A -85,B 0,C 180,E1 3406.517,E2 3406.517} C_VEL
LIN {X 0,Y 170.767,Z 1076.678,A -85,B 0,C 180,E1 3405.559,E2 3405.559} C_VEL
LIN {X 0,Y 166.973,Z 1094.182,A -85,B 0,C 180,E1 3404.748,E2 3404.748} C_VEL
LIN {X 0,Y 161.933,Z 1110.03,A -85,B 0,C 180,E1 3403.755,E2 3403.755} C_VEL
LIN {X 0,Y 155.201,Z 1125.916,A -85,B 0,C 180,E1 3402.438,E2 3402.438} C_VEL
LIN {X 0,Y 147.161,Z 1140.723,A -85,B 0,C 180,E1 3400.792,E2 3400.792} C_VEL
LIN {X 0,Y 138.211,Z 1154.121,A -85,B 0,C 180,E1 3398.794,E2 3398.794} C_VEL
LIN {X 0,Y 127.87,Z 1166.954,A -85,B 0,C 180,E1 3396.173,E2 3396.173} C_VEL
LIN {X 0,Y 116.837,Z 1178.427,A -85,B 0,C 180,E1 3392.861,E2 3392.861} C_VEL
LIN {X 0,Y 105.386,Z 1188.45,A -85,B 0,C 180,E1 3388.623,E2 3388.623} C_VEL
LIN {X 0,Y 93.059,Z 1197.521,A -85,B 0,C 180,E1 3382.65,E2 3382.65} C_VEL
LIN {X 0,Y 81.887,Z 1204.561,A -85,B 0,C 180,E1 3375.076,E2 3375.076} C_VEL
LIN {X 0,Y 71.847,Z 1210.083,A -85,B 0,C 180,E1 3364.778,E2 3364.778} C_VEL
LIN {X 0,Y 64.468,Z 1213.721,A -85,B 0,C 180,E1 3351.84,E2 3351.84} C_VEL
LIN {X 0,Y 60.495,Z 1215.758,A -85,B 0,C 180,E1 3335.678,E2 3335.678} C_VEL
LIN {X 0,Y 60.879,Z 1216.047,A -85,B 0,C 180,E1 3319.579,E2 3319.579} C_VEL
LIN {X 0,Y 65.643,Z 1214.608,A -85,B 0,C 180,E1 3303.772,E2 3303.772} C_VEL
LIN {X 0,Y 74.189,Z 1211.242,A -85,B 0,C 180,E1 3290.683,E2 3290.683} C_VEL
LIN {X 0,Y 78.023,Z 1209.522,A -85,B 0,C 180,E1 3286.535,E2 3286.535} C_VEL
LIN {X 0,Y 60.794,Z 1212.669,A -85,B 0,C 180,E1 3260.206,E2 3260.206} C_VEL
LIN {X 0,Y 58.879,Z 1213.599,A -85,B 0,C 180,E1 3250.767,E2 3250.767} C_VEL
LIN {X 0,Y 58.503,Z 1214.76,A -85,B 0,C 180,E1 3240.49,E2 3240.49} C_VEL
LIN {X 0,Y 59.562,Z 1221.218,A -85,B 0,C 180,E1 3227.394,E2 3227.394} C_VEL
LIN {X 0,Y 63.592,Z 1228.355,A -85,B 0,C 180,E1 3210.828,E2 3210.828} C_VEL
LIN {X 0,Y 72.858,Z 1235.324,A -85,B 0,C 180,E1 3194.863,E2 3194.863} C_VEL
LIN {X 0,Y 63.273,Z 1229.422,A -85,B 0,C 180,E1 3170.841,E2 3170.841} C_VEL
LIN {X 0,Y 61.531,Z 1230.667,A -85,B 0,C 180,E1 3155.608,E2 3155.608} C_VEL
LIN {X 0,Y 60.253,Z 1230.489,A -85,B 0,C 180,E1 3149.062,E2 3149.062} C_VEL
LIN {X 0,Y 58.948,Z 1228.693,A -85,B 0,C 180,E1 3132.237,E2 3132.237} C_VEL
LIN {X 0,Y 62.266,Z 1225.112,A -85,B 0,C 180,E1 3115.818,E2 3115.818} C_VEL
LIN {X 0,Y 69.84,Z 1219.637,A -85,B 0,C 180,E1 3101.903,E2 3101.903} C_VEL
LIN {X 0,Y 80.576,Z 1212.179,A -85,B 0,C 180,E1 3091.123,E2 3091.123} C_VEL
LIN {X 0,Y 92.666,Z 1203.128,A -85,B 0,C 180,E1 3083.508,E2 3083.508} C_VEL
LIN {X 0,Y 105.117,Z 1192.412,A -85,B 0,C 180,E1 3077.996,E2 3077.996} C_VEL
LIN {X 0,Y 117.44,Z 1180.127,A -85,B 0,C 180,E1 3073.959,E2 3073.959} C_VEL
LIN {X 0,Y 128.844,Z 1166.712,A -85,B 0,C 180,E1 3071.014,E2 3071.014} C_VEL
LIN {X 0,Y 139.129,Z 1152.121,A -85,B 0,C 180,E1 3068.83,E2 3068.83} C_VEL
LIN {X 0,Y 148.14,Z 1136.568,A -85,B 0,C 180,E1 3067.213,E2 3067.213} C_VEL
LIN {X 0,Y 155.331,Z 1121.077,A -85,B 0,C 180,E1 3066.046,E2 3066.046} C_VEL
LIN {X 0,Y 161.373,Z 1104.069,A -85,B 0,C 180,E1 3065.155,E2 3065.155} C_VEL
LIN {X 0,Y 165.676,Z 1086.687,A -85,B 0,C 180,E1 3064.553,E2 3064.553} C_VEL
LIN {X 0,Y 168.785,Z 1065.524,A -85,B 0,C 180,E1 3064.158,E2 3064.158} C_VEL
LIN {X 0,Y 172.613,Z 1033.721,A -85,B 0,C 180,E1 3063.823,E2 3063.823} C_VEL
LIN {X 0,Y 173.459,Z 1030.227,A -85,B 0,C 180,E1 3063.63,E2 3063.63} C_VEL
LIN {X 0,Y 173.98,Z 1027.058,A -85,B 0,C 180,E1 3063.007,E2 3063.007} C_VEL
LIN {X 0,Y 174.061,Z 1016.946,A -85,B 0,C 180,E1 3059.752,E2 3059.752} C_VEL
LIN {X 0,Y 174.323,Z 1014.239,A -85,B 0,C 180,E1 3059.227,E2 3059.227} C_VEL
LIN {X 0,Y 175.474,Z 1007.524,A -85,B 0,C 180,E1 3058.204,E2 3058.204} C_VEL
LIN {X 0,Y 183.771,Z 976.125,A -85,B 0,C 180,E1 3053.439,E2 3053.439} C_VEL
LIN {X 0,Y 190.594,Z 951.899,A -85,B 0,C 180,E1 3050.469,E2 3050.469} C_VEL
LIN {X 0,Y 186.543,Z 960.119,A -85,B 0,C 180,E1 3050.46,E2 3050.46} C_VEL
LIN {X 0,Y 181.657,Z 969.88,A -85,B 0,C 180,E1 3050.414,E2 3050.414} C_VEL
LIN {X 0,Y 172.723,Z 1047.023,A -85,B 0,C 180,E1 3049.07,E2 3049.07} C_VEL
LIN {X 0,Y 169.021,Z 1077.643,A -85,B 0,C 180,E1 3048.175,E2 3048.175} C_VEL
LIN {X 0,Y 165.127,Z 1095.127,A -85,B 0,C 180,E1 3047.416,E2 3047.416} C_VEL
LIN {X 0,Y 159.896,Z 1111.15,A -85,B 0,C 180,E1 3046.483,E2 3046.483} C_VEL
LIN {X 0,Y 152.996,Z 1127,A -85,B 0,C 180,E1 3045.271,E2 3045.271} C_VEL
LIN {X 0,Y 144.746,Z 1141.774,A -85,B 0,C 180,E1 3043.758,E2 3043.758} C_VEL
LIN {X 0,Y 134.746,Z 1156.197,A -85,B 0,C 180,E1 3041.753,E2 3041.753} C_VEL
LIN {X 0,Y 123.987,Z 1168.961,A -85,B 0,C 180,E1 3039.285,E2 3039.285} C_VEL
LIN {X 0,Y 112.57,Z 1180.243,A -85,B 0,C 180,E1 3036.171,E2 3036.171} C_VEL
LIN {X 0,Y 100.642,Z 1190.063,A -85,B 0,C 180,E1 3032.138,E2 3032.138} C_VEL
LIN {X 0,Y 87.683,Z 1199.009,A -85,B 0,C 180,E1 3026.334,E2 3026.334} C_VEL
LIN {X 0,Y 75.503,Z 1206.091,A -85,B 0,C 180,E1 3018.536,E2 3018.536} C_VEL
LIN {X 0,Y 64.904,Z 1211.304,A -85,B 0,C 180,E1 3008.025,E2 3008.025} C_VEL
LIN {X 0,Y 56.791,Z 1214.839,A -85,B 0,C 180,E1 2993.873,E2 2993.873} C_VEL
LIN {X 0,Y 52.494,Z 1216.783,A -85,B 0,C 180,E1 2975.45,E2 2975.45} C_VEL
LIN {X 0,Y 53.26,Z 1216.98,A -85,B 0,C 180,E1 2956.966,E2 2956.966} C_VEL
LIN {X 0,Y 58.611,Z 1215.55,A -85,B 0,C 180,E1 2940.333,E2 2940.333} C_VEL
LIN {X 0,Y 67.883,Z 1212.29,A -85,B 0,C 180,E1 2926.653,E2 2926.653} C_VEL
LIN {X 0,Y 53.302,Z 1215.026,A -85,B 0,C 180,E1 2902.036,E2 2902.036} C_VEL
LIN {X 0,Y 51.151,Z 1216.012,A -85,B 0,C 180,E1 2891.273,E2 2891.273} C_VEL
LIN {X 0,Y 50.699,Z 1217.152,A -85,B 0,C 180,E1 2878.87,E2 2878.87} C_VEL
LIN {X 0,Y 52.183,Z 1218.647,A -85,B 0,C 180,E1 2865.576,E2 2865.576} C_VEL
LIN {X 0,Y 56.283,Z 1225.216,A -85,B 0,C 180,E1 2848.989,E2 2848.989} C_VEL
LIN {X 0,Y 64.047,Z 1231.155,A -85,B 0,C 180,E1 2834.302,E2 2834.302} C_VEL
LIN {X 0,Y 57.512,Z 1227.693,A -85,B 0,C 180,E1 2819.146,E2 2819.146} C_VEL
LIN {X 0,Y 53.761,Z 1229.565,A -85,B 0,C 180,E1 2800.733,E2 2800.733} C_VEL
LIN {X 0,Y 53.537,Z 1229.74,A -85,B 0,C 180,E1 2795.373,E2 2795.373} C_VEL
LIN {X 0,Y 50.96,Z 1228.776,A -85,B 0,C 180,E1 2778.7,E2 2778.7} C_VEL
LIN {X 0,Y 52.847,Z 1226.023,A -85,B 0,C 180,E1 2759.297,E2 2759.297} C_VEL
LIN {X 0,Y 59.88,Z 1221.423,A -85,B 0,C 180,E1 2742.736,E2 2742.736} C_VEL
LIN {X 0,Y 70.646,Z 1214.917,A -85,B 0,C 180,E1 2730.326,E2 2730.326} C_VEL
LIN {X 0,Y 82.97,Z 1206.883,A -85,B 0,C 180,E1 2721.911,E2 2721.911} C_VEL
LIN {X 0,Y 95.726,Z 1197.369,A -85,B 0,C 180,E1 2716.093,E2 2716.093} C_VEL
LIN {X 0,Y 108.323,Z 1186.403,A -85,B 0,C 180,E1 2711.956,E2 2711.956} C_VEL
LIN {X 0,Y 120.416,Z 1173.995,A -85,B 0,C 180,E1 2708.883,E2 2708.883} C_VEL
LIN {X 0,Y 131.356,Z 1160.683,A -85,B 0,C 180,E1 2706.66,E2 2706.66} C_VEL
LIN {X 0,Y 141.009,Z 1146.562,A -85,B 0,C 180,E1 2705.014,E2 2705.014} C_VEL
LIN {X 0,Y 149.287,Z 1131.68,A -85,B 0,C 180,E1 2703.748,E2 2703.748} C_VEL
LIN {X 0,Y 156.652,Z 1114.98,A -85,B 0,C 180,E1 2702.787,E2 2702.787} C_VEL
LIN {X 0,Y 162.355,Z 1097.657,A -85,B 0,C 180,E1 2702.087,E2 2702.087} C_VEL
LIN {X 0,Y 166.193,Z 1080.367,A -85,B 0,C 180,E1 2701.679,E2 2701.679} C_VEL
LIN {X 0,Y 170.959,Z 1042.962,A -85,B 0,C 180,E1 2701.257,E2 2701.257} C_VEL
LIN {X 0,Y 172.3,Z 1031.996,A -85,B 0,C 180,E1 2701.203,E2 2701.203} C_VEL
LIN {X 0,Y 173.064,Z 1025.54,A -85,B 0,C 180,E1 2700.972,E2 2700.972} C_VEL
LIN {X 0,Y 174.323,Z 1014.239,A -85,B 0,C 180,E1 2699.227,E2 2699.227} C_VEL
LIN {X 0,Y 174.84,Z 1010.016,A -85,B 0,C 180,E1 2698.23,E2 2698.23} C_VEL
LIN {X 0,Y 176.403,Z 1000.987,A -85,B 0,C 180,E1 2694.56,E2 2694.56} C_VEL
LIN {X 0,Y 177.054,Z 997.317,A -85,B 0,C 180,E1 2693.746,E2 2693.746} C_VEL
LIN {X 0,Y 178.325,Z 989.644,A -85,B 0,C 180,E1 2692.658,E2 2692.658} C_VEL
LIN {X 0,Y 171.123,Z 1050.868,A -85,B 0,C 180,E1 2691.618,E2 2691.618} C_VEL
LIN {X 0,Y 167.577,Z 1078.912,A -85,B 0,C 180,E1 2690.829,E2 2690.829} C_VEL
LIN {X 0,Y 163.53,Z 1096.489,A -85,B 0,C 180,E1 2690.118,E2 2690.118} C_VEL
LIN {X 0,Y 158.23,Z 1112.269,A -85,B 0,C 180,E1 2689.276,E2 2689.276} C_VEL
LIN {X 0,Y 151.041,Z 1128.344,A -85,B 0,C 180,E1 2688.158,E2 2688.158} C_VEL
LIN {X 0,Y 142.262,Z 1143.538,A -85,B 0,C 180,E1 2686.739,E2 2686.739} C_VEL
LIN {X 0,Y 132.013,Z 1157.824,A -85,B 0,C 180,E1 2684.926,E2 2684.926} C_VEL
LIN {X 0,Y 120.493,Z 1170.96,A -85,B 0,C 180,E1 2682.588,E2 2682.588} C_VEL
LIN {X 0,Y 108.704,Z 1181.999,A -85,B 0,C 180,E1 2679.732,E2 2679.732} C_VEL
LIN {X 0,Y 95.443,Z 1192.291,A -85,B 0,C 180,E1 2675.683,E2 2675.683} C_VEL
LIN {X 0,Y 81.894,Z 1200.996,A -85,B 0,C 180,E1 2670.077,E2 2670.077} C_VEL
LIN {X 0,Y 69.29,Z 1207.649,A -85,B 0,C 180,E1 2662.511,E2 2662.511} C_VEL
LIN {X 0,Y 57.596,Z 1212.763,A -85,B 0,C 180,E1 2651.258,E2 2651.258} C_VEL
LIN {X 0,Y 48.406,Z 1216.265,A -85,B 0,C 180,E1 2634.383,E2 2634.383} C_VEL
LIN {X 0,Y 44.408,Z 1217.872,A -85,B 0,C 180,E1 2613.856,E2 2613.856} C_VEL
LIN {X 0,Y 46.037,Z 1217.838,A -85,B 0,C 180,E1 2592.28,E2 2592.28} C_VEL
LIN {X 0,Y 53.407,Z 1216.039,A -85,B 0,C 180,E1 2573.176,E2 2573.176} C_VEL
LIN {X 0,Y 57.724,Z 1214.744,A -85,B 0,C 180,E1 2566.68,E2 2566.68} C_VEL
LIN {X 0,Y 43.805,Z 1217.825,A -85,B 0,C 180,E1 2534.542,E2 2534.542} C_VEL
LIN {X 0,Y 42.921,Z 1219.254,A -85,B 0,C 180,E1 2517.33,E2 2517.33} C_VEL
LIN {X 0,Y 44.73,Z 1220.755,A -85,B 0,C 180,E1 2501.763,E2 2501.763} C_VEL
LIN {X 0,Y 50.807,Z 1223.488,A -85,B 0,C 180,E1 2482.404,E2 2482.404} C_VEL
LIN {X 0,Y 55.52,Z 1226.765,A -85,B 0,C 180,E1 2473.913,E2 2473.913} C_VEL
LIN {X 0,Y 53.21,Z 1225.757,A -85,B 0,C 180,E1 2469.032,E2 2469.032} C_VEL
LIN {X 0,Y 46.721,Z 1228.201,A -85,B 0,C 180,E1 2449.667,E2 2449.667} C_VEL
LIN {X 0,Y 45.506,Z 1228.774,A -85,B 0,C 180,E1 2436.325,E2 2436.325} C_VEL
LIN {X 0,Y 42.924,Z 1227.687,A -85,B 0,C 180,E1 2415.172,E2 2415.172} C_VEL
LIN {X 0,Y 46.293,Z 1224.779,A -85,B 0,C 180,E1 2392.809,E2 2392.809} C_VEL
LIN {X 0,Y 55.292,Z 1220.029,A -85,B 0,C 180,E1 2375.358,E2 2375.358} C_VEL
LIN {X 0,Y 67.719,Z 1213.393,A -85,B 0,C 180,E1 2363.495,E2 2363.495} C_VEL
LIN {X 0,Y 81.115,Z 1205.288,A -85,B 0,C 180,E1 2355.99,E2 2355.99} C_VEL
LIN {X 0,Y 94.683,Z 1195.587,A -85,B 0,C 180,E1 2350.9,E2 2350.9} C_VEL
LIN {X 0,Y 107.864,Z 1184.47,A -85,B 0,C 180,E1 2347.368,E2 2347.368} C_VEL
LIN {X 0,Y 119.906,Z 1172.414,A -85,B 0,C 180,E1 2344.879,E2 2344.879} C_VEL
LIN {X 0,Y 131.148,Z 1158.984,A -85,B 0,C 180,E1 2342.989,E2 2342.989} C_VEL
LIN {X 0,Y 141.023,Z 1144.639,A -85,B 0,C 180,E1 2341.588,E2 2341.588} C_VEL
LIN {X 0,Y 149.973,Z 1128.548,A -85,B 0,C 180,E1 2340.492,E2 2340.492} C_VEL
LIN {X 0,Y 156.968,Z 1112.563,A -85,B 0,C 180,E1 2339.763,E2 2339.763} C_VEL
LIN {X 0,Y 162.607,Z 1095.239,A -85,B 0,C 180,E1 2339.201,E2 2339.201} C_VEL
LIN {X 0,Y 166.34,Z 1077.761,A -85,B 0,C 180,E1 2338.859,E2 2338.859} C_VEL
LIN {X 0,Y 172.043,Z 1032.755,A -85,B 0,C 180,E1 2338.515,E2 2338.515} C_VEL
LIN {X 0,Y 172.693,Z 1027.484,A -85,B 0,C 180,E1 2338.341,E2 2338.341} C_VEL
LIN {X 0,Y 175.888,Z 1004.677,A -85,B 0,C 180,E1 2334.843,E2 2334.843} C_VEL
LIN {X 0,Y 177.054,Z 997.317,A -85,B 0,C 180,E1 2333.746,E2 2333.746} C_VEL
LIN {X 0,Y 176.625,Z 1000.726,A -85,B 0,C 180,E1 2333.78,E2 2333.78} C_VEL
LIN {X 0,Y 173.244,Z 1025.023,A -85,B 0,C 180,E1 2335.607,E2 2335.607} C_VEL
LIN {X 0,Y 172.025,Z 1034.672,A -85,B 0,C 180,E1 2335.818,E2 2335.818} C_VEL
LIN {X 0,Y 166.187,Z 1079.535,A -85,B 0,C 180,E1 2336.128,E2 2336.128} C_VEL
LIN {X 0,Y 162.044,Z 1097.045,A -85,B 0,C 180,E1 2336.408,E2 2336.408} C_VEL
LIN {X 0,Y 156.198,Z 1113.969,A -85,B 0,C 180,E1 2336.884,E2 2336.884} C_VEL
LIN {X 0,Y 148.609,Z 1130.451,A -85,B 0,C 180,E1 2337.506,E2 2337.506} C_VEL
LIN {X 0,Y 139.573,Z 1145.824,A -85,B 0,C 180,E1 2338.405,E2 2338.405} C_VEL
LIN {X 0,Y 128.973,Z 1160.392,A -85,B 0,C 180,E1 2339.633,E2 2339.633} C_VEL
LIN {X 0,Y 117.002,Z 1173.948,A -85,B 0,C 180,E1 2341.293,E2 2341.293} C_VEL
LIN {X 0,Y 104.171,Z 1186.036,A -85,B 0,C 180,E1 2343.534,E2 2343.534} C_VEL
LIN {X 0,Y 90.581,Z 1196.656,A -85,B 0,C 180,E1 2346.633,E2 2346.633} C_VEL
LIN {X 0,Y 76.08,Z 1206.114,A -85,B 0,C 180,E1 2351.37,E2 2351.37} C_VEL
LIN {X 0,Y 61.291,Z 1214.169,A -85,B 0,C 180,E1 2358.921,E2 2358.921} C_VEL
LIN {X 0,Y 47.935,Z 1220.346,A -85,B 0,C 180,E1 2371.247,E2 2371.247} C_VEL
LIN {X 0,Y 38.18,Z 1224.595,A -85,B 0,C 180,E1 2391.086,E2 2391.086} C_VEL
LIN {X 0,Y 35.076,Z 1227.186,A -85,B 0,C 180,E1 2420.174,E2 2420.174} C_VEL
LIN {X 0,Y 37.775,Z 1227.8,A -85,B 0,C 180,E1 2439.159,E2 2439.159} C_VEL
LIN {X 0,Y 41.324,Z 1226.591,A -85,B 0,C 180,E1 2462.184,E2 2462.184} C_VEL
LIN {X 0,Y 45.943,Z 1225.093,A -85,B 0,C 180,E1 2473.606,E2 2473.606} C_VEL
LIN {X 0,Y 40.47,Z 1223.619,A -85,B 0,C 180,E1 2485.371,E2 2485.371} C_VEL
LIN {X 0,Y 36.332,Z 1221.819,A -85,B 0,C 180,E1 2504.026,E2 2504.026} C_VEL
LIN {X 0,Y 35.043,Z 1220.282,A -85,B 0,C 180,E1 2524.911,E2 2524.911} C_VEL
LIN {X 0,Y 41.153,Z 1218.033,A -85,B 0,C 180,E1 2555.671,E2 2555.671} C_VEL
LIN {X 0,Y 47.434,Z 1216.944,A -85,B 0,C 180,E1 2567.149,E2 2567.149} C_VEL
LIN {X 0,Y 38.87,Z 1218.724,A -85,B 0,C 180,E1 2587.282,E2 2587.282} C_VEL
LIN {X 0,Y 36.408,Z 1218.86,A -85,B 0,C 180,E1 2613.127,E2 2613.127} C_VEL
LIN {X 0,Y 40.856,Z 1217.383,A -85,B 0,C 180,E1 2637.688,E2 2637.688} C_VEL
LIN {X 0,Y 51.202,Z 1213.979,A -85,B 0,C 180,E1 2656.242,E2 2656.242} C_VEL
LIN {X 0,Y 63.955,Z 1208.967,A -85,B 0,C 180,E1 2667.567,E2 2667.567} C_VEL
LIN {X 0,Y 77.413,Z 1202.438,A -85,B 0,C 180,E1 2674.771,E2 2674.771} C_VEL
LIN {X 0,Y 91.553,Z 1193.904,A -85,B 0,C 180,E1 2679.897,E2 2679.897} C_VEL
LIN {X 0,Y 105.289,Z 1183.753,A -85,B 0,C 180,E1 2683.54,E2 2683.54} C_VEL
LIN {X 0,Y 117.421,Z 1172.885,A -85,B 0,C 180,E1 2686.079,E2 2686.079} C_VEL
LIN {X 0,Y 128.753,Z 1160.629,A -85,B 0,C 180,E1 2688.067,E2 2688.067} C_VEL
LIN {X 0,Y 139.222,Z 1146.731,A -85,B 0,C 180,E1 2689.678,E2 2689.678} C_VEL
LIN {X 0,Y 148.311,Z 1131.798,A -85,B 0,C 180,E1 2690.957,E2 2690.957} C_VEL
LIN {X 0,Y 155.99,Z 1115.803,A -85,B 0,C 180,E1 2691.989,E2 2691.989} C_VEL
LIN {X 0,Y 161.956,Z 1099.055,A -85,B 0,C 180,E1 2692.817,E2 2692.817} C_VEL
LIN {X 0,Y 166.289,Z 1081.258,A -85,B 0,C 180,E1 2693.488,E2 2693.488} C_VEL
LIN {X 0,Y 169.405,Z 1058.656,A -85,B 0,C 180,E1 2694.115,E2 2694.115} C_VEL
LIN {X 0,Y 173.558,Z 1023.63,A -85,B 0,C 180,E1 2694.831,E2 2694.831} C_VEL
LIN {X 0,Y 172.505,Z 1030.754,A -85,B 0,C 180,E1 2695.83,E2 2695.83} C_VEL
LIN {X 0,Y 172.025,Z 1034.672,A -85,B 0,C 180,E1 2695.818,E2 2695.818} C_VEL
LIN {X 0,Y 172.01,Z 1034.926,A -85,B 0,C 180,E1 2695.816,E2 2695.816} C_VEL
LIN {X 0,Y 172.01,Z 1141.92,A -85,B 0,C 180,E1 2695.816,E2 2695.816} C_VEL
LIN {X 0,Y 155.583,Z 1141.92,A -85,B 0,C 180,E1 2694.907,E2 2694.907} C_VEL
LIN {X 0,Y 153.611,Z 1139.92,A -85,B 0,C 180,E1 2694.785,E2 2694.785} C_VEL
LIN {X 0,Y 153.611,Z 1128.585,A -85,B 0,C 180,E1 2694.785,E2 2694.785} C_VEL
LIN {X 0,Y 150.044,Z 1127.649,A -85,B 0,C 180,E1 2694.327,E2 2694.327} C_VEL
LIN {X 0,Y 141.429,Z 1142.717,A -85,B 0,C 180,E1 2693.324,E2 2693.324} C_VEL
LIN {X 0,Y 131.224,Z 1156.94,A -85,B 0,C 180,E1 2692.072,E2 2692.072} C_VEL
LIN {X 0,Y 119.62,Z 1170.059,A -85,B 0,C 180,E1 2690.479,E2 2690.479} C_VEL
LIN {X 0,Y 107.138,Z 1181.653,A -85,B 0,C 180,E1 2688.462,E2 2688.462} C_VEL
LIN {X 0,Y 93.84,Z 1191.809,A -85,B 0,C 180,E1 2685.806,E2 2685.806} C_VEL
LIN {X 0,Y 79.832,Z 1200.483,A -85,B 0,C 180,E1 2682.121,E2 2682.121} C_VEL
LIN {X 0,Y 65.33,Z 1207.708,A -85,B 0,C 180,E1 2676.648,E2 2676.648} C_VEL
LIN {X 0,Y 50.818,Z 1213.408,A -85,B 0,C 180,E1 2667.756,E2 2667.756} C_VEL
LIN {X 0,Y 38.196,Z 1217.27,A -85,B 0,C 180,E1 2652.863,E2 2652.863} C_VEL
LIN {X 0,Y 29.523,Z 1219.457,A -85,B 0,C 180,E1 2625.693,E2 2625.693} C_VEL
LIN {X 0,Y 29.849,Z 1219.873,A -85,B 0,C 180,E1 2590.401,E2 2590.401} C_VEL
LIN {X 0,Y 37.006,Z 1218.849,A -85,B 0,C 180,E1 2567.228,E2 2567.228} C_VEL
LIN {X 0,Y 27.632,Z 1221.063,A -85,B 0,C 180,E1 2534.673,E2 2534.673} C_VEL
LIN {X 0,Y 27.25,Z 1222.211,A -85,B 0,C 180,E1 2513.68,E2 2513.68} C_VEL
LIN {X 0,Y 29.367,Z 1223.313,A -85,B 0,C 180,E1 2495.885,E2 2495.885} C_VEL
LIN {X 0,Y 36.33,Z 1225.264,A -85,B 0,C 180,E1 2473.114,E2 2473.114} C_VEL
LIN {X 0,Y 29.993,Z 1226.803,A -85,B 0,C 180,E1 2443.522,E2 2443.522} C_VEL
LIN {X 0,Y 28.118,Z 1226.67,A -85,B 0,C 180,E1 2432.066,E2 2432.066} C_VEL
LIN {X 0,Y 28.545,Z 1224.986,A -85,B 0,C 180,E1 2395.947,E2 2395.947} C_VEL
LIN {X 0,Y 37.984,Z 1221.561,A -85,B 0,C 180,E1 2369.737,E2 2369.737} C_VEL
LIN {X 0,Y 51.875,Z 1216.302,A -85,B 0,C 180,E1 2355.533,E2 2355.533} C_VEL
LIN {X 0,Y 67.213,Z 1209.206,A -85,B 0,C 180,E1 2347.694,E2 2347.694} C_VEL
LIN {X 0,Y 83.083,Z 1200.184,A -85,B 0,C 180,E1 2342.905,E2 2342.905} C_VEL
LIN {X 0,Y 97.974,Z 1189.798,A -85,B 0,C 180,E1 2339.891,E2 2339.891} C_VEL
LIN {X 0,Y 112.053,Z 1177.788,A -85,B 0,C 180,E1 2337.82,E2 2337.82} C_VEL
LIN {X 0,Y 124.718,Z 1164.727,A -85,B 0,C 180,E1 2336.395,E2 2336.395} C_VEL
LIN {X 0,Y 135.401,Z 1151.415,A -85,B 0,C 180,E1 2335.425,E2 2335.425} C_VEL
LIN {X 0,Y 145.095,Z 1136.672,A -85,B 0,C 180,E1 2334.674,E2 2334.674} C_VEL
LIN {X 0,Y 150.044,Z 1127.649,A -85,B 0,C 180,E1 2334.327,E2 2334.327} C_VEL
LIN {X 0,Y 153.791,Z 1128.561,A -85,B 0,C 180,E1 2334.139,E2 2334.139} C_VEL
LIN {X 0,Y 153.791,Z 1187.302,A -85,B 0,C 180,E1 2334.139,E2 2334.139} C_VEL
LIN {X 0,Y 117.952,Z 1187.302,A -85,B 0,C 180,E1 2334.194,E2 2334.194} C_VEL
LIN {X 0,Y 115.952,Z 1185.302,A -85,B 0,C 180,E1 2334.198,E2 2334.198} C_VEL
LIN {X 0,Y 115.952,Z 1178.063,A -85,B 0,C 180,E1 2334.198,E2 2334.198} C_VEL
LIN {X 0,Y 112.876,Z 1176.54,A -85,B 0,C 180,E1 2333.603,E2 2333.603} C_VEL
LIN {X 0,Y 99.986,Z 1187.261,A -85,B 0,C 180,E1 2331.842,E2 2331.842} C_VEL
LIN {X 0,Y 85.448,Z 1197.113,A -85,B 0,C 180,E1 2329.348,E2 2329.348} C_VEL
LIN {X 0,Y 70.142,Z 1205.321,A -85,B 0,C 180,E1 2325.731,E2 2325.731} C_VEL
LIN {X 0,Y 54.278,Z 1211.947,A -85,B 0,C 180,E1 2319.923,E2 2319.923} C_VEL
LIN {X 0,Y 39.274,Z 1216.652,A -85,B 0,C 180,E1 2309.912,E2 2309.912} C_VEL
LIN {X 0,Y 26.5,Z 1219.551,A -85,B 0,C 180,E1 2289.86,E2 2289.86} C_VEL
LIN {X 0,Y 20.447,Z 1220.839,A -85,B 0,C 180,E1 2247.159,E2 2247.159} C_VEL
LIN {X 0,Y 26.66,Z 1220.446,A -85,B 0,C 180,E1 2207.781,E2 2207.781} C_VEL
LIN {X 0,Y 19.256,Z 1222.955,A -85,B 0,C 180,E1 2154.039,E2 2154.039} C_VEL
LIN {X 0,Y 22.255,Z 1224.176,A -85,B 0,C 180,E1 2127.375,E2 2127.375} C_VEL
LIN {X 0,Y 26.273,Z 1225.17,A -85,B 0,C 180,E1 2111.736,E2 2111.736} C_VEL
LIN {X 0,Y 21.941,Z 1225.861,A -85,B 0,C 180,E1 2085.905,E2 2085.905} C_VEL
LIN {X 0,Y 20.037,Z 1224.702,A -85,B 0,C 180,E1 2036.754,E2 2036.754} C_VEL
LIN {X 0,Y 30.437,Z 1221.744,A -85,B 0,C 180,E1 2003.163,E2 2003.163} C_VEL
LIN {X 0,Y 45.619,Z 1216.965,A -85,B 0,C 180,E1 1988.825,E2 1988.825} C_VEL
LIN {X 0,Y 62.069,Z 1210.33,A -85,B 0,C 180,E1 1981.846,E2 1981.846} C_VEL
LIN {X 0,Y 78.021,Z 1202.167,A -85,B 0,C 180,E1 1978.066,E2 1978.066} C_VEL
LIN {X 0,Y 93.243,Z 1192.437,A -85,B 0,C 180,E1 1975.653,E2 1975.653} C_VEL
LIN {X 0,Y 107.55,Z 1181.293,A -85,B 0,C 180,E1 1974.064,E2 1974.064} C_VEL
LIN {X 0,Y 112.876,Z 1176.54,A -85,B 0,C 180,E1 1973.603,E2 1973.603} C_VEL
LIN {X 0,Y 116.19,Z 1178.014,A -85,B 0,C 180,E1 1973.349,E2 1973.349} C_VEL
LIN {X 0,Y 116.19,Z 1214.685,A -85,B 0,C 180,E1 1973.349,E2 1973.349} C_VEL
LIN {X 0,Y 76.59,Z 1214.685,A -85,B 0,C 180,E1 1973.491,E2 1973.491} C_VEL
LIN {X 0,Y 74.59,Z 1212.685,A -85,B 0,C 180,E1 1973.503,E2 1973.503} C_VEL
LIN {X 0,Y 74.59,Z 1206.595,A -85,B 0,C 180,E1 1973.503,E2 1973.503} C_VEL
LIN {X 0,Y 71.888,Z 1204.788,A -85,B 0,C 180,E1 1972.78,E2 1972.78} C_VEL
LIN {X 0,Y 55.954,Z 1211.562,A -85,B 0,C 180,E1 1969.289,E2 1969.289} C_VEL
LIN {X 0,Y 39.692,Z 1216.65,A -85,B 0,C 180,E1 1963.121,E2 1963.121} C_VEL
LIN {X 0,Y 23.476,Z 1220.123,A -85,B 0,C 180,E1 1948.347,E2 1948.347} C_VEL
LIN {X 0,Y 12.885,Z 1221.697,A -85,B 0,C 180,E1 1903.4,E2 1903.4} C_VEL
LIN {X 0,Y 15.948,Z 1221.792,A -85,B 0,C 180,E1 1848.795,E2 1848.795} C_VEL
LIN {X 0,Y 11.536,Z 1223.573,A -85,B 0,C 180,E1 1784.929,E2 1784.929} C_VEL
LIN {X 0,Y 15.423,Z 1224.538,A -85,B 0,C 180,E1 1754.507,E2 1754.507} C_VEL
LIN {X 0,Y 16.319,Z 1224.748,A -85,B 0,C 180,E1 1749.173,E2 1749.173} C_VEL
LIN {X 0,Y 14.278,Z 1224.885,A -85,B 0,C 180,E1 1734.905,E2 1734.905} C_VEL
LIN {X 0,Y 13.885,Z 1223.704,A -85,B 0,C 180,E1 1657.708,E2 1657.708} C_VEL
LIN {X 0,Y 28.221,Z 1220.731,A -85,B 0,C 180,E1 1627.452,E2 1627.452} C_VEL
LIN {X 0,Y 45,Z 1215.976,A -85,B 0,C 180,E1 1618.334,E2 1618.334} C_VEL
LIN {X 0,Y 62.3,Z 1209.326,A -85,B 0,C 180,E1 1614.18,E2 1614.18} C_VEL
LIN {X 0,Y 71.888,Z 1204.788,A -85,B 0,C 180,E1 1612.78,E2 1612.78} C_VEL
LIN {X 0,Y 74.783,Z 1206.559,A -85,B 0,C 180,E1 1612.428,E2 1612.428} C_VEL
LIN {X 0,Y 74.783,Z 1229.963,A -85,B 0,C 180,E1 1612.428,E2 1612.428} C_VEL
LIN {X 0,Y 30.831,Z 1229.963,A -85,B 0,C 180,E1 1612.156,E2 1612.156} C_VEL
LIN {X 0,Y 28.831,Z 1227.963,A -85,B 0,C 180,E1 1612.124,E2 1612.124} C_VEL
LIN {X 0,Y 28.831,Z 1222.098,A -85,B 0,C 180,E1 1612.124,E2 1612.124} C_VEL
LIN {X 0,Y 26.576,Z 1220.123,A -85,B 0,C 180,E1 1611.014,E2 1611.014} C_VEL
LIN {X 0,Y 10.09,Z 1222.264,A -85,B 0,C 180,E1 1592.942,E2 1592.942} C_VEL
LIN {X 0,Y 5.154,Z 1222.823,A -85,B 0,C 180,E1 1495.551,E2 1495.551} C_VEL
LIN {X 0,Y 5.067,Z 1223.822,A -85,B 0,C 180,E1 1387.258,E2 1387.258} C_VEL
LIN {X 0,Y 13.998,Z 1222.274,A -85,B 0,C 180,E1 1257.478,E2 1257.478} C_VEL
LIN {X 0,Y 26.576,Z 1220.123,A -85,B 0,C 180,E1 1251.014,E2 1251.014} C_VEL
LIN {X 0,Y 28.95,Z 1222.084,A -85,B 0,C 180,E1 1250.393,E2 1250.393} C_VEL
LIN {X 0,Y 28.95,Z 1305,A -85,B 0,C 180,E1 1250.393,E2 1250.393} C_VEL
LIN {X 0,Y 28.95,Z 1305,A -85,B 0,C 180,E1 1250.393,E2 1250.393}

QRS_NEXT_CUT()

QRS_NEXT()
QRS_HOME()

END
